# EPICS substitutions: viocs/bo_ps/bo_psApp/Db/kickers.substitutions
file "db/kickers.db" {
    pattern { family, pos }
        { "KICKERINJ", "01D" }
        { "KICKEREXT", "48D-A"}
        { "KICKEREXT", "48D-B"}
}
